{attribute 'no_explicit_call' := 'do not call this POU directly'}
// Store arguments in a single string seperated by $R
FUNCTION_BLOCK FB_Argument IMPLEMENTS I_Argument
VAR_INPUT
END_VAR
VAR_OUTPUT
END_VAR
VAR
	sValue:					STRING(255);		// storage for arguments
END_VAR
(*
    Tc3_Event – TwinCAT 3 Event Logging Framework
    Copyright (c) Peter Zerlauth

    This component is provided under a Dual Licensing Model:

    1. GPLv3 Open-Source License
       - Free for personal, educational, and non-commercial use.
       - Commercial use allowed only if the entire application is published
         under GPLv3, including all modifications to this code.
       - Requires full disclosure of source code for derivative works.

    2. Commercial License
       - Required for integration into proprietary or closed-source products.
       - Removes all GPLv3 copyleft obligations.
       - Includes optional warranty, professional support, and long-term
         maintenance options.

    For commercial licensing, contact:
        info@peterzerlauth.com

    By using this Function Block you agree to the terms of the selected license.
*)

// add boolean value to arguments
METHOD PUBLIC M_AddBOOL : I_Argument
VAR_INPUT
	bValue:				BOOL;		// Boolean input value
END_VAR
sValue:= CONCAT(sValue, BOOL_TO_STRING(bValue));			// convert
sValue:= CONCAT(sValue, '$R');								// add separator
M_AddBOOL:= THIS^;
END_METHOD

// add int value to arguments
METHOD PUBLIC M_AddINT : I_Argument
VAR_INPUT
	nValue:				LINT;		// Integer input value
END_VAR
VAR
	sTemp: 			STRING;
END_VAR
sValue:= CONCAT(sValue, CONCAT(LINT_TO_STRING(nValue), '$R'));	// add new arg
M_AddINT:= THIS^;
END_METHOD

// add real value to arguments
METHOD PUBLIC M_AddREAL : I_Argument
VAR_INPUT
	fValue:				LREAL;		// Real input value
	nDecimals:			USINT;		// Decimals afer .
END_VAR
VAR
	sTemp: 			STRING;
END_VAR
sValue:= CONCAT(sValue, CONCAT(LREAL_TO_FMTSTR(fValue, nDecimals, TRUE), '$R'));				// add new arg
M_AddREAL:= THIS^;
END_METHOD

// add string value to arguments
METHOD PUBLIC M_AddSTRING : I_Argument
VAR_INPUT
	sValue:				STRING(255);		// String input value
END_VAR
THIS^.sValue:= CONCAT(THIS^.sValue, CONCAT(sValue, '$R'));				// add separator 
M_AddSTRING:= THIS^;
END_METHOD

// add time value to arguments
METHOD PUBLIC M_AddTIME : I_Argument
VAR_INPUT
	tValue:				TIME;		// Time input value
END_VAR
sValue:= CONCAT(sValue, CONCAT(TIME_TO_STRING(tValue), '$R'));				// add separator
M_AddTIME:= THIS^;
END_METHOD

// Clear arguments
METHOD PUBLIC M_Clear : I_Argument
VAR_INPUT
END_VAR
sValue:= '';
M_Clear:= THIS^;
END_METHOD

// Returns the list with arguments
PROPERTY PUBLIC P_Value : STRING(255)
GET
P_Value:= sValue;
END_GET
END_PROPERTY

END_FUNCTION_BLOCK

(* stored: Version 1.1.0.1
   POU FB_Argument: Id {a8de1bab-544f-463d-b649-c52e572fc35a}, SpecialFunc None
   Method M_AddBOOL: Id {6fe5c2f5-9f6f-45ef-a512-7b981b0be320}
   Method M_AddINT: Id {0fb61d34-2130-4e2b-8ca3-a66334bd442e}
   Method M_AddREAL: Id {ec2078de-d198-403e-9f1d-9aa3713c42cf}
   Method M_AddSTRING: Id {6ddea08b-8528-414a-b8b0-ca7a04ccfa78}
   Method M_AddTIME: Id {5bf7bbc0-6a06-4191-858d-e9e3e764bb18}
   Method M_Clear: Id {1a899f54-f4aa-43d6-ba56-2488949d893d}
   Property P_Value: Id {364579c4-8829-400e-a5c9-b1603a0f22c8}
   Get Get: Id {a740fb78-092e-4273-9e56-34b846282910} *)
